# EPICS substitutions: pgpCamlinkApp/camera_config/Jai_GO_5000M_PMCL_UV.substitutions
# A simple MODEL substitutions file which preserves macro defaults
# but expands any inluded rbvMonitor.template or other templates.
file Jai_GO_5000M_PMCL_UV.template
{
	{
		P				= "\$(P)",
		R				= "\$(R)",
		PORT			= "\$(PORT)",
		PWIDTH			= "\$(PWIDTH=TRIG:PULSE:WIDTH)",
		PW_SCALE		= "\$(PW_SCALE=1e6)",
	}
}
